TYPE "MES_Msg"
VERSION : 0.1
// Block: MES_Msg
   STRUCT
      Id : DInt;
      timestamp : String;
      topic : UDInt;
      payLoad : String;
   END_STRUCT;

END_TYPE
